(* IEC 61131-3 sources: codesys-mcp-toolkit/standalone-sync/sources_st/511_05/Util/FB_InfluxBuffer, 4 files *)

(* ---- FB_InfluxBuffer.fb.st ---- *)
// @OBJECT_ID: d2828cf0-a55e-4108-8a78-43bc321d9b6a
// @DECLARATION
FUNCTION_BLOCK FB_InfluxBuffer
VAR_INPUT
    sMeasurement : STRING(80);   // Measurement name (e.g., 'CEX6')
    sTagKey      : STRING(40);   // Tag name (e.g., 'title')
    sTagValue    : STRING(80);   // Tag value (e.g., 'kolonna_23b')
END_VAR

VAR_OUTPUT
    sBuffer      : STRING(5000); // Resulting string for fbSender
END_VAR

VAR
    iCurrentLen  : INT;          // Current length of sBuffer
END_VAR

// @IMPLEMENTATION
// Initialization: Clear buffer and add Measurement + Tag
// Format: "Measurement,TagKey=TagValue " (note the space at the end)
sBuffer := CONCAT(sMeasurement, ',');
sBuffer := CONCAT(sBuffer, sTagKey);
sBuffer := CONCAT(sBuffer, '=');
sBuffer := CONCAT(sBuffer, sTagValue);
sBuffer := CONCAT(sBuffer, ' '); // Line protocol space between tags and fields

iCurrentLen := LEN(sBuffer);

(* ---- AddDword.method.st ---- *)
// @OBJECT_ID: a5b3bcec-b63f-42e1-9ad1-aa88a7512f3d
// @DECLARATION
METHOD PUBLIC AddDWord : BOOL
VAR_INPUT
    sName : STRING(40);
    dwVal : DWORD;
END_VAR
VAR
    sFragment : STRING(100);
    sTemp     : STRING(20);
END_VAR

// @IMPLEMENTATION

// Add comma if not the first field
IF iCurrentLen > (LEN(sMeasurement) + LEN(sTagKey) + LEN(sTagValue) + 3) THEN
    sFragment := ',';
ELSE
    sFragment := '';
END_IF

// Format: Key=Value (DWORD преобразуется в UDINT для строки)
sFragment := CONCAT(sFragment, sName);
sFragment := CONCAT(sFragment, '=');

// Convert DWORD to string
sTemp := DWORD_TO_STRING(dwVal);
sFragment := CONCAT(sFragment, sTemp);

// Append to buffer
STU.StrConcatA(ADR(sFragment), ADR(sBuffer), SIZEOF(sBuffer));
iCurrentLen := LEN(sBuffer);
AddDWord := TRUE;

(* ---- AddReal.method.st ---- *)
// @OBJECT_ID: 0f7dc9ff-fcad-4997-a2b3-68e2ac3befdf
// @DECLARATION
METHOD PUBLIC AddReal : BOOL
VAR_INPUT
    sName : STRING(40);
    rVal  : REAL;
END_VAR
VAR
    sFragment : STRING(100);
END_VAR

// @IMPLEMENTATION

// Add comma if not the first field
IF iCurrentLen > (LEN(sMeasurement) + LEN(sTagKey) + LEN(sTagValue) + 3) THEN
    sFragment := ',';
ELSE
    sFragment := '';
END_IF

// Format: Key=Value
sFragment := CONCAT(sFragment, sName);
sFragment := CONCAT(sFragment, '=');
sFragment := CONCAT(sFragment, REAL_TO_STRING(rVal));

// Append to buffer using STU for safety or simple CONCAT
STU.StrConcatA(ADR(sFragment), ADR(sBuffer), SIZEOF(sBuffer));
iCurrentLen := LEN(sBuffer);
AddReal := TRUE;

(* ---- Clear.method.st ---- *)
// @OBJECT_ID: 5ef3d038-d9c2-4048-9196-bfdb9bff4938
// @DECLARATION
METHOD Clear : BOOL
VAR_INPUT
END_VAR

// @IMPLEMENTATION
// Очистка буфера для нового измерения
sBuffer := CONCAT(sMeasurement, ',');
sBuffer := CONCAT(sBuffer, sTagKey);
sBuffer := CONCAT(sBuffer, '=');
sBuffer := CONCAT(sBuffer, sTagValue);
sBuffer := CONCAT(sBuffer, ' ');

iCurrentLen := LEN(sBuffer);
Clear := TRUE;
